FUNCTION_BLOCK FB_ProfileCheckMeasure
VAR_INPUT
	LastBeamBlocked		: UINT;
	Offset 				: INT; 
	BeamSpacing 		: INT;
	StartMeasurement	: BOOL;
END_VAR

VAR
ConvertedLastBeamBlocked		: INT;
TempMeasuredValue : INT;
END_VAR

VAR_OUTPUT
	MaxMeasuredValue 	: INT;
	LiveValue			: INT;
	LightGridClear		: BOOL;
END_VAR

//65535(uint) = -1 (int) = no beams blocked
ConvertedLastBeamBlocked:= UINT_TO_INT(LastBeamBlocked);

IF ConvertedLastBeamBlocked >= 0 THEN
	LiveValue := (ConvertedLastBeamBlocked * BeamSpacing) - Offset;	
ELSE
	LiveValue := 0;	
END_IF
	
IF StartMeasurement THEN 
	IF LiveValue > MaxMeasuredValue THEN
		MaxMeasuredValue := LiveValue;
	END_IF
ELSE 
	MaxMeasuredValue := 0;
END_IF

IF (ConvertedLastBeamBlocked = -1) THEN
	LightGridClear := TRUE;
ELSE
	LightGridClear := FALSE;	
END_IF

END_FUNCTION_BLOCK

(* stored: Version 1.1.0.1, ProductVersion 3.1.4024.9
   POU FB_ProfileCheckMeasure: Id {0ca37436-616f-41aa-9f72-ea12d8a1ad68}, SpecialFunc None *)
